TYPE ST_SafeDiag_HardwareInfos :
STRUCT
	iVoltageC1				: INT;		// CoE - F985:01	[mV]	
	iVoltageC2				: INT;		// CoE - F984:01	[mV]		
	iTemperatureC1			: INT;		// CoE - F984:02	[Celcius degrees]   
	iTemperatureC2			: INT;		// CoE - F985:02    [Celcius degrees]
END_STRUCT
END_TYPE

(* stored: Version 1.1.0.1, ProductVersion 3.1.4024.12
   DUT ST_SafeDiag_HardwareInfos: Id {e6678f16-c359-47d9-ba9f-43e7b55499d0} *)
